FUNCTION_BLOCK Generator (* Service Interface Function Block Type *)
  (* Standard: 61499-2 *)
  (* Version 1.0, 2024-12-18, cochicde *)
  PACKAGE performance;
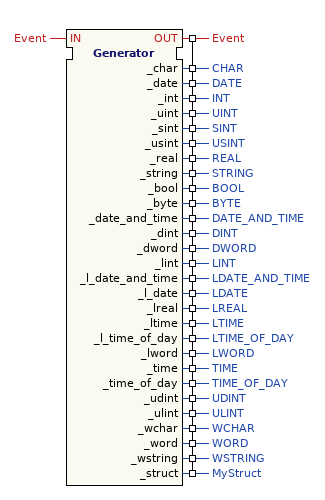
  EVENT_INPUT
    IN; (* Service Initialization *)
  END_EVENT
  EVENT_OUTPUT
    OUT WITH _char, _date, _int, _uint, _sint, _usint, _real, _string, _bool, _byte, _date_and_time, _dint, _dword, _lint, _l_date_and_time, _l_date, _lreal, _ltime, _l_time_of_day, _lword, _time, _time_of_day, _udint, _ulint, _wchar, _word, _wstring, _struct; (* Initialization Confirm *)
  END_EVENT
  VAR_OUTPUT
    _char : CHAR; (* Event Output Qualifier *)
    _date : DATE; (* Service Status *)
    _int : INT; (* Input data from resource *)
    _uint : UINT;
    _sint : SINT;
    _usint : USINT;
    _real : REAL;
    _string : STRING;
    _bool : BOOL;
    _byte : BYTE;
    _date_and_time : DATE_AND_TIME;
    _dint : DINT;
    _dword : DWORD;
    _lint : LINT;
    _l_date_and_time : LDATE_AND_TIME;
    _l_date : LDATE;
    _lreal : LREAL;
    _ltime : LTIME;
    _l_time_of_day : LTIME_OF_DAY;
    _lword : LWORD;
    _time : TIME;
    _time_of_day : TIME_OF_DAY;
    _udint : UDINT;
    _ulint : ULINT;
    _wchar : WCHAR;
    _word : WORD;
    _wstring : WSTRING;
    _struct : MyStruct; {SET_ATTRIBUTE(VarConfig, false)}
  END_VAR
  SERVICE APPLICATION/RESOURCE (* Service Interface Function Block Type *)
    SEQUENCE normal_establishment
      APPLICATION.INIT+(PARAMS) -> RESOURCE.initialize(PARAMS) -> APPLICATION.INITO+();
    END_SEQUENCE
    SEQUENCE unsuccessful_establishment
      APPLICATION.INIT+(PARAMS) -> RESOURCE.initialize(PARAMS) -> APPLICATION.INITO-(STATUS);
    END_SEQUENCE
    SEQUENCE request_confirm
      APPLICATION.REQ+(SD) -> RESOURCE.request(SD) -> APPLICATION.CNF+(RD);
    END_SEQUENCE
    SEQUENCE request_inhibited
      APPLICATION.REQ-(SD) -> APPLICATION.CNF-(STATUS);
    END_SEQUENCE
    SEQUENCE request_error
      APPLICATION.REQ+(SD) -> RESOURCE.request(SD) -> APPLICATION.CNF-(STATUS);
    END_SEQUENCE
    SEQUENCE indication_response
      RESOURCE.indicate(RD) -> APPLICATION.IND+(RD);
      APPLICATION.RSP(QI,SD) -> RESOURCE.response(QI,SD);
    END_SEQUENCE
    SEQUENCE indication_inhibited
      RESOURCE.indicate(RD,QI=FALSE) -> RESOURCE.inhibited();
    END_SEQUENCE
    SEQUENCE error_indication
      RESOURCE.error(STATUS) -> APPLICATION.IND-(STATUS);
    END_SEQUENCE
    SEQUENCE application_initiated_termination
      APPLICATION.INIT-() -> RESOURCE.terminate() -> APPLICATION.INITO-(STATUS);
    END_SEQUENCE
    SEQUENCE resource_initiated_termination
      -> APPLICATION.INITO-(STATUS);
    END_SEQUENCE
  END_SERVICE
END_FUNCTION_BLOCK
